// vecA*=num
FUNCTION vecSelfMultiNum : BOOL
VAR_IN_OUT 
	vecA :ARRAY[*] OF LREAL;
END_VAR

VAR_INPUT
	num :LREAL;
END_VAR

VAR
	m :DINT;
	i :DINT;
 
END_VAR

m:=UPPER_BOUND(vecA,1);

FOR i:=1 TO m DO
		vecA[i]:=num*vecA[i];
END_FOR

END_FUNCTION

(* stored: Version 1.1.0.1, ProductVersion 3.1.4024.11
   POU vecSelfMultiNum: Id {8965e60b-9e28-4b9c-9ec6-21311af54a9f}, SpecialFunc None *)
